DATA_BLOCK "ST10Cylinder"
{ S7_Optimized_Access := 'FALSE' }
VERSION : 0.1
// ATTRIBUTES
// AUTO_NUMBER = False
// BLOCK_NUMBER = 1020
// END_ATTRIBUTES
   STRUCT
      Cy : Array[1..110] of "Cyl";
   END_STRUCT;


BEGIN
   Cy[1].In.Error := false;
   Cy[1].In.GoWorkInterlock := false;
   Cy[1].In.GoHomeInterlock := false;
   Cy[1].In.WorkPositionSensor := false;
   Cy[1].In.HomePositionSensor := false;
   Cy[1].In.ValveType := false;
   Cy[1].In.ManualOutputType := false;
   Cy[1].In.FaultTime := 50;
   Cy[1].In.OnPositionTime := 10;
   Cy[1].Inout.ManualGoWork := FALSE;
   Cy[1].Inout.ManualGoHome := FALSE;
   Cy[1].Inout.AutoGoWork := FALSE;
   Cy[1].Inout.AutoGoHome := FALSE;
   Cy[1].S.GoWorkTime := 0;
   Cy[1].S.GoHomeTime := 0;
   Cy[1].S.WorkFaultTime := 0;
   Cy[1].S.HomeFaultTime := 0;
   Cy[1].S.BothSensorOnTime := 0;
   Cy[1].S.Pulse100mSP := FALSE;
   Cy[1].S.AutoGoWorkP := FALSE;
   Cy[1].S.AutoGoHomeP := FALSE;
   Cy[1].S.GoWork100mSP := TRUE;
   Cy[1].S.GoHome100mSP := TRUE;
   Cy[1].S.BothSensorOn100mSP := TRUE;
   Cy[1].S.Alarm := FALSE;
   Cy[1].S.spare1 := FALSE;
   Cy[1].S.spare2 := 16#00;
   Cy[1].Out.GoWorkPosition := FALSE;
   Cy[1].Out.GoHomePosition := FALSE;
   Cy[1].Out.GoWPButtonActive := TRUE;
   Cy[1].Out.GoHPButtonActive := TRUE;
   Cy[1].Out.GoWorkFault := FALSE;
   Cy[1].Out.GoHomeFault := FALSE;
   Cy[1].Out.SensorPositionFault := FALSE;
   Cy[1].Out.CyNO := 16#01;
   Cy[2].In.Error := false;
   Cy[2].In.GoWorkInterlock := false;
   Cy[2].In.GoHomeInterlock := false;
   Cy[2].In.WorkPositionSensor := false;
   Cy[2].In.HomePositionSensor := false;
   Cy[2].In.ValveType := true;
   Cy[2].In.ManualOutputType := false;
   Cy[2].In.FaultTime := 50;
   Cy[2].In.OnPositionTime := 10;
   Cy[2].Inout.ManualGoWork := FALSE;
   Cy[2].Inout.ManualGoHome := FALSE;
   Cy[2].Inout.AutoGoWork := FALSE;
   Cy[2].Inout.AutoGoHome := FALSE;
   Cy[2].S.GoWorkTime := 0;
   Cy[2].S.GoHomeTime := 0;
   Cy[2].S.WorkFaultTime := 0;
   Cy[2].S.HomeFaultTime := 0;
   Cy[2].S.BothSensorOnTime := 0;
   Cy[2].S.Pulse100mSP := FALSE;
   Cy[2].S.AutoGoWorkP := FALSE;
   Cy[2].S.AutoGoHomeP := FALSE;
   Cy[2].S.GoWork100mSP := TRUE;
   Cy[2].S.GoHome100mSP := TRUE;
   Cy[2].S.BothSensorOn100mSP := TRUE;
   Cy[2].S.Alarm := FALSE;
   Cy[2].S.spare1 := FALSE;
   Cy[2].S.spare2 := 16#00;
   Cy[2].Out.GoWorkPosition := FALSE;
   Cy[2].Out.GoHomePosition := TRUE;
   Cy[2].Out.GoWPButtonActive := TRUE;
   Cy[2].Out.GoHPButtonActive := TRUE;
   Cy[2].Out.GoWorkFault := FALSE;
   Cy[2].Out.GoHomeFault := FALSE;
   Cy[2].Out.SensorPositionFault := FALSE;
   Cy[2].Out.CyNO := 16#02;
   Cy[3].In.Error := false;
   Cy[3].In.GoWorkInterlock := false;
   Cy[3].In.GoHomeInterlock := false;
   Cy[3].In.WorkPositionSensor := false;
   Cy[3].In.HomePositionSensor := false;
   Cy[3].In.ValveType := false;
   Cy[3].In.ManualOutputType := false;
   Cy[3].In.FaultTime := 50;
   Cy[3].In.OnPositionTime := 10;
   Cy[3].Inout.ManualGoWork := FALSE;
   Cy[3].Inout.ManualGoHome := FALSE;
   Cy[3].Inout.AutoGoWork := FALSE;
   Cy[3].Inout.AutoGoHome := FALSE;
   Cy[3].S.GoWorkTime := 0;
   Cy[3].S.GoHomeTime := 0;
   Cy[3].S.WorkFaultTime := 0;
   Cy[3].S.HomeFaultTime := 0;
   Cy[3].S.BothSensorOnTime := 0;
   Cy[3].S.Pulse100mSP := FALSE;
   Cy[3].S.AutoGoWorkP := FALSE;
   Cy[3].S.AutoGoHomeP := FALSE;
   Cy[3].S.GoWork100mSP := TRUE;
   Cy[3].S.GoHome100mSP := TRUE;
   Cy[3].S.BothSensorOn100mSP := TRUE;
   Cy[3].S.Alarm := FALSE;
   Cy[3].S.spare1 := FALSE;
   Cy[3].S.spare2 := 16#00;
   Cy[3].Out.GoWorkPosition := FALSE;
   Cy[3].Out.GoHomePosition := FALSE;
   Cy[3].Out.GoWPButtonActive := TRUE;
   Cy[3].Out.GoHPButtonActive := TRUE;
   Cy[3].Out.GoWorkFault := FALSE;
   Cy[3].Out.GoHomeFault := FALSE;
   Cy[3].Out.SensorPositionFault := FALSE;
   Cy[3].Out.CyNO := 16#03;
   Cy[4].In.Error := false;
   Cy[4].In.GoWorkInterlock := false;
   Cy[4].In.GoHomeInterlock := false;
   Cy[4].In.WorkPositionSensor := false;
   Cy[4].In.HomePositionSensor := false;
   Cy[4].In.ValveType := true;
   Cy[4].In.ManualOutputType := false;
   Cy[4].In.FaultTime := 50;
   Cy[4].In.OnPositionTime := 10;
   Cy[4].Inout.ManualGoWork := FALSE;
   Cy[4].Inout.ManualGoHome := FALSE;
   Cy[4].Inout.AutoGoWork := FALSE;
   Cy[4].Inout.AutoGoHome := FALSE;
   Cy[4].S.GoWorkTime := 0;
   Cy[4].S.GoHomeTime := 0;
   Cy[4].S.WorkFaultTime := 0;
   Cy[4].S.HomeFaultTime := 0;
   Cy[4].S.BothSensorOnTime := 0;
   Cy[4].S.Pulse100mSP := FALSE;
   Cy[4].S.AutoGoWorkP := FALSE;
   Cy[4].S.AutoGoHomeP := FALSE;
   Cy[4].S.GoWork100mSP := TRUE;
   Cy[4].S.GoHome100mSP := TRUE;
   Cy[4].S.BothSensorOn100mSP := TRUE;
   Cy[4].S.Alarm := FALSE;
   Cy[4].S.spare1 := FALSE;
   Cy[4].S.spare2 := 16#00;
   Cy[4].Out.GoWorkPosition := FALSE;
   Cy[4].Out.GoHomePosition := TRUE;
   Cy[4].Out.GoWPButtonActive := TRUE;
   Cy[4].Out.GoHPButtonActive := TRUE;
   Cy[4].Out.GoWorkFault := FALSE;
   Cy[4].Out.GoHomeFault := FALSE;
   Cy[4].Out.SensorPositionFault := FALSE;
   Cy[4].Out.CyNO := 16#04;
   Cy[5].In.Error := false;
   Cy[5].In.GoWorkInterlock := false;
   Cy[5].In.GoHomeInterlock := false;
   Cy[5].In.WorkPositionSensor := false;
   Cy[5].In.HomePositionSensor := false;
   Cy[5].In.ValveType := false;
   Cy[5].In.ManualOutputType := false;
   Cy[5].In.FaultTime := 50;
   Cy[5].In.OnPositionTime := 10;
   Cy[5].Inout.ManualGoWork := FALSE;
   Cy[5].Inout.ManualGoHome := FALSE;
   Cy[5].Inout.AutoGoWork := FALSE;
   Cy[5].Inout.AutoGoHome := FALSE;
   Cy[5].S.GoWorkTime := 0;
   Cy[5].S.GoHomeTime := 0;
   Cy[5].S.WorkFaultTime := 0;
   Cy[5].S.HomeFaultTime := 0;
   Cy[5].S.BothSensorOnTime := 0;
   Cy[5].S.Pulse100mSP := FALSE;
   Cy[5].S.AutoGoWorkP := FALSE;
   Cy[5].S.AutoGoHomeP := FALSE;
   Cy[5].S.GoWork100mSP := TRUE;
   Cy[5].S.GoHome100mSP := TRUE;
   Cy[5].S.BothSensorOn100mSP := TRUE;
   Cy[5].S.Alarm := FALSE;
   Cy[5].S.spare1 := FALSE;
   Cy[5].S.spare2 := 16#00;
   Cy[5].Out.GoWorkPosition := FALSE;
   Cy[5].Out.GoHomePosition := FALSE;
   Cy[5].Out.GoWPButtonActive := TRUE;
   Cy[5].Out.GoHPButtonActive := TRUE;
   Cy[5].Out.GoWorkFault := FALSE;
   Cy[5].Out.GoHomeFault := FALSE;
   Cy[5].Out.SensorPositionFault := FALSE;
   Cy[5].Out.CyNO := 16#05;
   Cy[6].In.Error := false;
   Cy[6].In.GoWorkInterlock := false;
   Cy[6].In.GoHomeInterlock := false;
   Cy[6].In.WorkPositionSensor := false;
   Cy[6].In.HomePositionSensor := false;
   Cy[6].In.ValveType := true;
   Cy[6].In.ManualOutputType := false;
   Cy[6].In.FaultTime := 50;
   Cy[6].In.OnPositionTime := 10;
   Cy[6].Inout.ManualGoWork := FALSE;
   Cy[6].Inout.ManualGoHome := FALSE;
   Cy[6].Inout.AutoGoWork := FALSE;
   Cy[6].Inout.AutoGoHome := FALSE;
   Cy[6].S.GoWorkTime := 0;
   Cy[6].S.GoHomeTime := 0;
   Cy[6].S.WorkFaultTime := 0;
   Cy[6].S.HomeFaultTime := 0;
   Cy[6].S.BothSensorOnTime := 0;
   Cy[6].S.Pulse100mSP := FALSE;
   Cy[6].S.AutoGoWorkP := FALSE;
   Cy[6].S.AutoGoHomeP := FALSE;
   Cy[6].S.GoWork100mSP := TRUE;
   Cy[6].S.GoHome100mSP := TRUE;
   Cy[6].S.BothSensorOn100mSP := TRUE;
   Cy[6].S.Alarm := FALSE;
   Cy[6].S.spare1 := FALSE;
   Cy[6].S.spare2 := 16#00;
   Cy[6].Out.GoWorkPosition := FALSE;
   Cy[6].Out.GoHomePosition := FALSE;
   Cy[6].Out.GoWPButtonActive := TRUE;
   Cy[6].Out.GoHPButtonActive := TRUE;
   Cy[6].Out.GoWorkFault := FALSE;
   Cy[6].Out.GoHomeFault := FALSE;
   Cy[6].Out.SensorPositionFault := FALSE;
   Cy[6].Out.CyNO := 16#06;
   Cy[7].In.Error := false;
   Cy[7].In.GoWorkInterlock := false;
   Cy[7].In.GoHomeInterlock := false;
   Cy[7].In.WorkPositionSensor := false;
   Cy[7].In.HomePositionSensor := false;
   Cy[7].In.ValveType := true;
   Cy[7].In.ManualOutputType := false;
   Cy[7].In.FaultTime := 50;
   Cy[7].In.OnPositionTime := 10;
   Cy[7].Inout.ManualGoWork := FALSE;
   Cy[7].Inout.ManualGoHome := FALSE;
   Cy[7].Inout.AutoGoWork := FALSE;
   Cy[7].Inout.AutoGoHome := FALSE;
   Cy[7].S.GoWorkTime := 0;
   Cy[7].S.GoHomeTime := 0;
   Cy[7].S.WorkFaultTime := 0;
   Cy[7].S.HomeFaultTime := 0;
   Cy[7].S.BothSensorOnTime := 0;
   Cy[7].S.Pulse100mSP := FALSE;
   Cy[7].S.AutoGoWorkP := FALSE;
   Cy[7].S.AutoGoHomeP := FALSE;
   Cy[7].S.GoWork100mSP := TRUE;
   Cy[7].S.GoHome100mSP := TRUE;
   Cy[7].S.BothSensorOn100mSP := TRUE;
   Cy[7].S.Alarm := FALSE;
   Cy[7].S.spare1 := FALSE;
   Cy[7].S.spare2 := 16#00;
   Cy[7].Out.GoWorkPosition := FALSE;
   Cy[7].Out.GoHomePosition := FALSE;
   Cy[7].Out.GoWPButtonActive := TRUE;
   Cy[7].Out.GoHPButtonActive := TRUE;
   Cy[7].Out.GoWorkFault := FALSE;
   Cy[7].Out.GoHomeFault := FALSE;
   Cy[7].Out.SensorPositionFault := FALSE;
   Cy[7].Out.CyNO := 16#07;
   Cy[8].In.Error := false;
   Cy[8].In.GoWorkInterlock := false;
   Cy[8].In.GoHomeInterlock := false;
   Cy[8].In.WorkPositionSensor := false;
   Cy[8].In.HomePositionSensor := false;
   Cy[8].In.ValveType := true;
   Cy[8].In.ManualOutputType := false;
   Cy[8].In.FaultTime := 50;
   Cy[8].In.OnPositionTime := 10;
   Cy[8].Inout.ManualGoWork := FALSE;
   Cy[8].Inout.ManualGoHome := FALSE;
   Cy[8].Inout.AutoGoWork := FALSE;
   Cy[8].Inout.AutoGoHome := FALSE;
   Cy[8].S.GoWorkTime := 0;
   Cy[8].S.GoHomeTime := 0;
   Cy[8].S.WorkFaultTime := 0;
   Cy[8].S.HomeFaultTime := 0;
   Cy[8].S.BothSensorOnTime := 0;
   Cy[8].S.Pulse100mSP := FALSE;
   Cy[8].S.AutoGoWorkP := FALSE;
   Cy[8].S.AutoGoHomeP := FALSE;
   Cy[8].S.GoWork100mSP := TRUE;
   Cy[8].S.GoHome100mSP := TRUE;
   Cy[8].S.BothSensorOn100mSP := TRUE;
   Cy[8].S.Alarm := FALSE;
   Cy[8].S.spare1 := FALSE;
   Cy[8].S.spare2 := 16#00;
   Cy[8].Out.GoWorkPosition := FALSE;
   Cy[8].Out.GoHomePosition := FALSE;
   Cy[8].Out.GoWPButtonActive := TRUE;
   Cy[8].Out.GoHPButtonActive := TRUE;
   Cy[8].Out.GoWorkFault := FALSE;
   Cy[8].Out.GoHomeFault := FALSE;
   Cy[8].Out.SensorPositionFault := FALSE;
   Cy[8].Out.CyNO := 16#08;
   Cy[9].In.Error := false;
   Cy[9].In.GoWorkInterlock := false;
   Cy[9].In.GoHomeInterlock := false;
   Cy[9].In.WorkPositionSensor := false;
   Cy[9].In.HomePositionSensor := false;
   Cy[9].In.ValveType := true;
   Cy[9].In.ManualOutputType := false;
   Cy[9].In.FaultTime := 50;
   Cy[9].In.OnPositionTime := 10;
   Cy[9].Inout.ManualGoWork := FALSE;
   Cy[9].Inout.ManualGoHome := FALSE;
   Cy[9].Inout.AutoGoWork := FALSE;
   Cy[9].Inout.AutoGoHome := FALSE;
   Cy[9].S.GoWorkTime := 0;
   Cy[9].S.GoHomeTime := 0;
   Cy[9].S.WorkFaultTime := 0;
   Cy[9].S.HomeFaultTime := 0;
   Cy[9].S.BothSensorOnTime := 0;
   Cy[9].S.Pulse100mSP := FALSE;
   Cy[9].S.AutoGoWorkP := FALSE;
   Cy[9].S.AutoGoHomeP := FALSE;
   Cy[9].S.GoWork100mSP := TRUE;
   Cy[9].S.GoHome100mSP := TRUE;
   Cy[9].S.BothSensorOn100mSP := TRUE;
   Cy[9].S.Alarm := FALSE;
   Cy[9].S.spare1 := FALSE;
   Cy[9].S.spare2 := 16#00;
   Cy[9].Out.GoWorkPosition := FALSE;
   Cy[9].Out.GoHomePosition := FALSE;
   Cy[9].Out.GoWPButtonActive := TRUE;
   Cy[9].Out.GoHPButtonActive := TRUE;
   Cy[9].Out.GoWorkFault := FALSE;
   Cy[9].Out.GoHomeFault := FALSE;
   Cy[9].Out.SensorPositionFault := FALSE;
   Cy[9].Out.CyNO := 16#09;
   Cy[10].In.Error := false;
   Cy[10].In.GoWorkInterlock := false;
   Cy[10].In.GoHomeInterlock := false;
   Cy[10].In.WorkPositionSensor := false;
   Cy[10].In.HomePositionSensor := false;
   Cy[10].In.ValveType := true;
   Cy[10].In.ManualOutputType := false;
   Cy[10].In.FaultTime := 50;
   Cy[10].In.OnPositionTime := 10;
   Cy[10].Inout.ManualGoWork := FALSE;
   Cy[10].Inout.ManualGoHome := FALSE;
   Cy[10].Inout.AutoGoWork := FALSE;
   Cy[10].Inout.AutoGoHome := FALSE;
   Cy[10].S.GoWorkTime := 0;
   Cy[10].S.GoHomeTime := 0;
   Cy[10].S.WorkFaultTime := 0;
   Cy[10].S.HomeFaultTime := 0;
   Cy[10].S.BothSensorOnTime := 0;
   Cy[10].S.Pulse100mSP := FALSE;
   Cy[10].S.AutoGoWorkP := FALSE;
   Cy[10].S.AutoGoHomeP := FALSE;
   Cy[10].S.GoWork100mSP := TRUE;
   Cy[10].S.GoHome100mSP := TRUE;
   Cy[10].S.BothSensorOn100mSP := TRUE;
   Cy[10].S.Alarm := FALSE;
   Cy[10].S.spare1 := FALSE;
   Cy[10].S.spare2 := 16#00;
   Cy[10].Out.GoWorkPosition := FALSE;
   Cy[10].Out.GoHomePosition := FALSE;
   Cy[10].Out.GoWPButtonActive := FALSE;
   Cy[10].Out.GoHPButtonActive := FALSE;
   Cy[10].Out.GoWorkFault := FALSE;
   Cy[10].Out.GoHomeFault := FALSE;
   Cy[10].Out.SensorPositionFault := FALSE;
   Cy[10].Out.CyNO := 16#0A;

END_DATA_BLOCK

